(* IEC 61131-3 sources: Industry-PLC-LLM/data/PLCBEAD_repo/PLCBEAD_PLCEmbed-main/PLC-BEAD/Source/GEB/ACOSH, 1 file *)

(* ---- ACOSH.ST ---- *)
FUNCTION ACOSH:REAL
	VAR_INPUT
		X :	REAL;
	END_VAR
	ACOSH := LN(SQRT(X * X - 1.0) + X);

END_FUNCTION

PROGRAM program0
  VAR
    LocalVar0 : REAL;
    LocalOUT  : REAL;
  END_VAR

  LocalOUT := ACOSH(LocalVar0);
END_PROGRAM
